{attribute 'linkalways'} 
{attribute 'no_explicit_call' := 'This FB is a CLASS and must be accessed using methods or properties'}
{attribute 'enable_dynamic_creation'}
FUNCTION_BLOCK _ETcVnOcrModelType EXTENDS EnumDatatypeBase
VAR
	localData : ETcVnOcrModelType;
	activeData : REFERENCE TO ETcVnOcrModelType;
	enumBaseDatatype : _ULINT(localData);
END_VAR

METHOD PRIVATE AddLocalEnumeration
VAR_INPUT
	Enumeration : T_MAXSTRING;
	Value : ETcVnOcrModelType;
END_VAR
AddEnumeration(Enumeration, Value);
END_METHOD

PROPERTY PUBLIC Address : PVOID
GET
Address := ADR(activeData);
END_GET
END_PROPERTY

METHOD PUBLIC ClearReference
VAR_INPUT
END_VAR
activeData REF= localData;
SetBaseDatatypeReference();
END_METHOD

METHOD PUBLIC Clone : I_Datatype
VAR
    pClone : POINTER TO _ETcVnOcrModelType;
END_VAR
pClone := __NEW(_ETcVnOcrModelType(InitialValue := Value));
Clone := pClone^;
END_METHOD

METHOD FB_init : BOOL
VAR_INPUT
	bInitRetains : BOOL; // if TRUE, the retain variables are initialized (warm start / cold start)
	bInCopyCode : BOOL;  // if TRUE, the instance afterwards gets moved into the copy code (online change)
	InitialValue : ETcVnOcrModelType;
END_VAR
localData := InitialValue;
AddBaseDatatype(enumBaseDatatype);
ClearReference();

AddLocalEnumeration('TCVN_OMT_NUMBERS', ETcVnOcrModelType.TCVN_OMT_NUMBERS);
AddLocalEnumeration('TCVN_OMT_NUMBERS_SC', ETcVnOcrModelType.TCVN_OMT_NUMBERS_SC);
AddLocalEnumeration('TCVN_OMT_UCLETTERS', ETcVnOcrModelType.TCVN_OMT_UCLETTERS);
AddLocalEnumeration('TCVN_OMT_NUMBERS_SC_UCLETTERS', ETcVnOcrModelType.TCVN_OMT_NUMBERS_SC_UCLETTERS);
END_METHOD

PROPERTY PUBLIC Identifier : T_MAXSTRING
GET
Identifier := 'ETcVnOcrModelType';
END_GET
END_PROPERTY

METHOD IsEnumeratorValueEqual : BOOL
VAR_INPUT
	Enumerator : I_KeyValueForwardEnumerator;
END_VAR
VAR
	storedValue : ETcVnOcrModelType;
END_VAR
IF NOT Enumerator.TryGet(storedValue) THEN
	RETURN;
END_IF

IsEnumeratorValueEqual := storedValue = activeData;
END_METHOD

METHOD PUBLIC MakeReferenceTo
VAR_INPUT
	ReferenceTarget : REFERENCE TO ETcVnOcrModelType;
END_VAR
activeData REF= ReferenceTarget;
SetBaseDatatypeReference();
END_METHOD

METHOD PROTECTED SetBaseDatatypeReference
VAR_INPUT
END_VAR
enumBaseDatatype.MakeReferenceTo(activeData);
END_METHOD

PROPERTY PUBLIC Size : UDINT
GET
Size := SIZEOF(activeData);
END_GET
END_PROPERTY

METHOD TryMakeReferenceTo : BOOL
VAR_INPUT
	Target : I_Datatype;
END_VAR
VAR
	targetAsEnum : I_EnumDatatype;
	pTargetData : POINTER TO ETcVnOcrModelType;
END_VAR
IF NOT Target.TryResolveAsEnumDatatype(targetAsEnum) THEN
	RETURN;
END_IF

IF targetAsEnum.Identifier <> Identifier THEN
	RETURN;
END_IF

pTargetData := Target.Address;
activeData REF= pTargetData^;
SetBaseDatatypeReference();
TryMakeReferenceTo := TRUE;
END_METHOD

PROPERTY PUBLIC Value : ETcVnOcrModelType
GET
Value := activeData;
END_GET
SET
activeData := Value;
END_SET
END_PROPERTY

END_FUNCTION_BLOCK

(* stored: Version 1.1.0.1, ProductVersion 3.1.4024.12
   POU _ETcVnOcrModelType: Id {abceaebb-d705-4e06-b536-e9a4428f9a9a}, SpecialFunc None
   Folder Constructor: Id {7ed1025b-c417-4e58-a0fb-e18c80f851a8}
   Folder Private: Id {fef7c9b5-add5-46b0-90c4-03723892aa77}
   Folder Protected: Id {89b28910-4b0a-4068-9e31-060090c2b558}
   Method AddLocalEnumeration: Id {eea7d105-2e70-417f-b1c3-b9ab5e838280}
   Property Address: Id {e6cd3c9e-5949-41f4-bcd0-16aa3b881f2a}
   Get Get: Id {3db69e9d-d6b3-46a8-8ff8-3cbb70c41fb2}
   Method ClearReference: Id {86c97a40-2db7-4054-b3a7-a279562f7e80}
   Method Clone: Id {361bb9d9-4403-4feb-b0b4-47ea6023f6d6}
   Method FB_init: Id {e087a28b-0d5c-4432-901d-98af72f0a9f0}
   Property Identifier: Id {bed293f0-8128-49e0-ae7e-ad7a81c66a74}
   Get Get: Id {845332c7-1f2c-4442-9c5d-69a28221bd51}
   Method IsEnumeratorValueEqual: Id {29bd07ad-6b28-46d2-beac-192bc4cd6a75}
   Method MakeReferenceTo: Id {60bf9aff-f737-4be3-9a9b-b47e91e5ab1c}
   Method SetBaseDatatypeReference: Id {223f75ff-f511-41a1-bb27-724f3e7cfd64}
   Property Size: Id {b8a2d8e1-eaa7-4552-8914-037d0296b6d6}
   Get Get: Id {f6962b78-5aaf-48ad-b19e-8c3749f49778}
   Method TryMakeReferenceTo: Id {d7e8979c-e994-4878-96ad-f80879977a99}
   Property Value: Id {fc9f9193-7351-4bff-8def-c2881c24e2e4}
   Get Get: Id {42454915-6b8b-444c-898f-aefbc63841c2}
   Set Set: Id {3cbca391-0dc4-44fb-9571-76f643398b9d} *)
